{attribute 'qualified_only'}
TYPE E_PlayerID :
(
	player1 := 4,
    player2 := 10,
    player3 := 21,
    player4 := 27,
    all := 31
) INT;
END_TYPE

(* stored: Version 1.1.0.1, ProductVersion 3.1.4024.9
   DUT E_PlayerID: Id {fba0b20b-516a-456c-a5e5-ca35d88970e7} *)
